// TIA Portal V18 export
// export: Created 2026-06-24T03:56:38.2149864Z, ExportSetting WithDefaults, DisplayName Totally Integrated Automation Portal, DisplayVersion V18, DisplayName TIA Portal Openness, DisplayVersion V18, DisplayName TIA Portal Version Control Interface, DisplayVersion V18, DisplayName STEP 7 Professional, DisplayVersion V18, DisplayName STEP 7 Safety, DisplayVersion V18, DisplayName WinCC Professional, DisplayVersion V18
DATA_BLOCK "PI_DB"   // DB3
VERSION : 0.1
// stored: AutoNumber true, InstanceOfName PID, InstanceOfType FB
"PID"
   // VAR_INPUT
   //    ki : Real;
   //    kp : Real;
   //    kd : Real;
   //    level : Real;
   //    setpoint : Real;
   //    drain : Bool;
   //    "full drain" : Bool;
   //    emergency : Bool;
   // END_VAR
   // VAR_OUTPUT
   //    filling : Real;
   //    draining : Real;
   //    errordisplay : Real;
   //    setpointdisplay : DInt;
   //    leveldisplay : DInt;
   // END_VAR
   // VAR
   //    integralop : Real;
   //    oldintegral : Real;
   //    err2 : Real;
   // END_VAR
BEGIN
END_DATA_BLOCK
